SUBAPPLICATION Uebung_177_AX (* Beispiel für AX_FB_R_TRIG (Rising Edge Detection) *)
  (* Standard: 61499-2; Description: Copyright (c) 2023 Meisterschulen am Ostbahnhof This program and the accompanying materials are made available under the terms of the Eclipse Public License 2.0 which is available at https://www.eclipse.org/legal/epl-2.0/ SPDX-License-Identifier: EPL-2.0 *)
  (* Version 1.0, 2025-02-01, Franz Höpfinger, Meisterschulen am Ostbahnhof, initial API and implementation and/or initial documentation *)
  PACKAGE Uebungen;
  IMPORT logiBUS::io::DI::logiBUS_DI::Input_I1;
  IMPORT logiBUS::io::DQ::logiBUS_DO::Output_Q1;
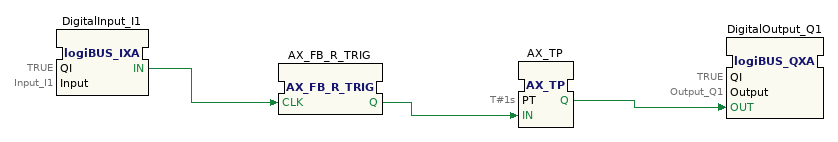
  FBS
    AX_FB_R_TRIG : adapter::iec61131::edgeDetection::AX_FB_R_TRIG;
    DigitalOutput_Q1 : logiBUS::io::DQ::logiBUS_QXA(QI := TRUE, Output := Output_Q1);
    DigitalInput_I1 : logiBUS::io::DI::logiBUS_IXA(QI := TRUE, Input := Input_I1);
    AX_TP : adapter::events::unidirectional::timers::AX_TP(PT := T#1s);
  END_FBS
  ADAPTER_CONNECTIONS
    DigitalInput_I1.IN TO AX_FB_R_TRIG.CLK;
    AX_TP.Q TO DigitalOutput_Q1.OUT;
    AX_FB_R_TRIG.Q TO AX_TP.IN;
  END_CONNECTIONS
END_SUBAPPLICATION
